FUNCTION_BLOCK MANUAL_PAGE
VAR_INPUT
	STRING_PG1 : STRING;
	STRING_PG2 : STRING;
	STRING_PG3 : STRING;
	STRING_PG4 : STRING;
	STRING_PG5 : STRING;
	STRING_PG6 : STRING;
	STRING_PG7 : STRING;
	STRING_PG8 : STRING;
	STRING_PG9 : STRING;
	STRING_PG10 : STRING;
	STRING_PG11 : STRING;
	STRING_PG12 : STRING;
	STRING_PG13 : STRING;
	STRING_PG14 : STRING;
	STRING_PG15 : STRING;
	STRING_PG16 : STRING;
	STRING_PG17 : STRING;
	STRING_PG18 : STRING;
	STRING_PG19 : STRING;
	STRING_PG20 : STRING;
	STRING_CVISU : STRING;


END_VAR
VAR_OUTPUT
	PG_CONFIRMED_BOOL : BOOL;

END_VAR
VAR
END_VAR

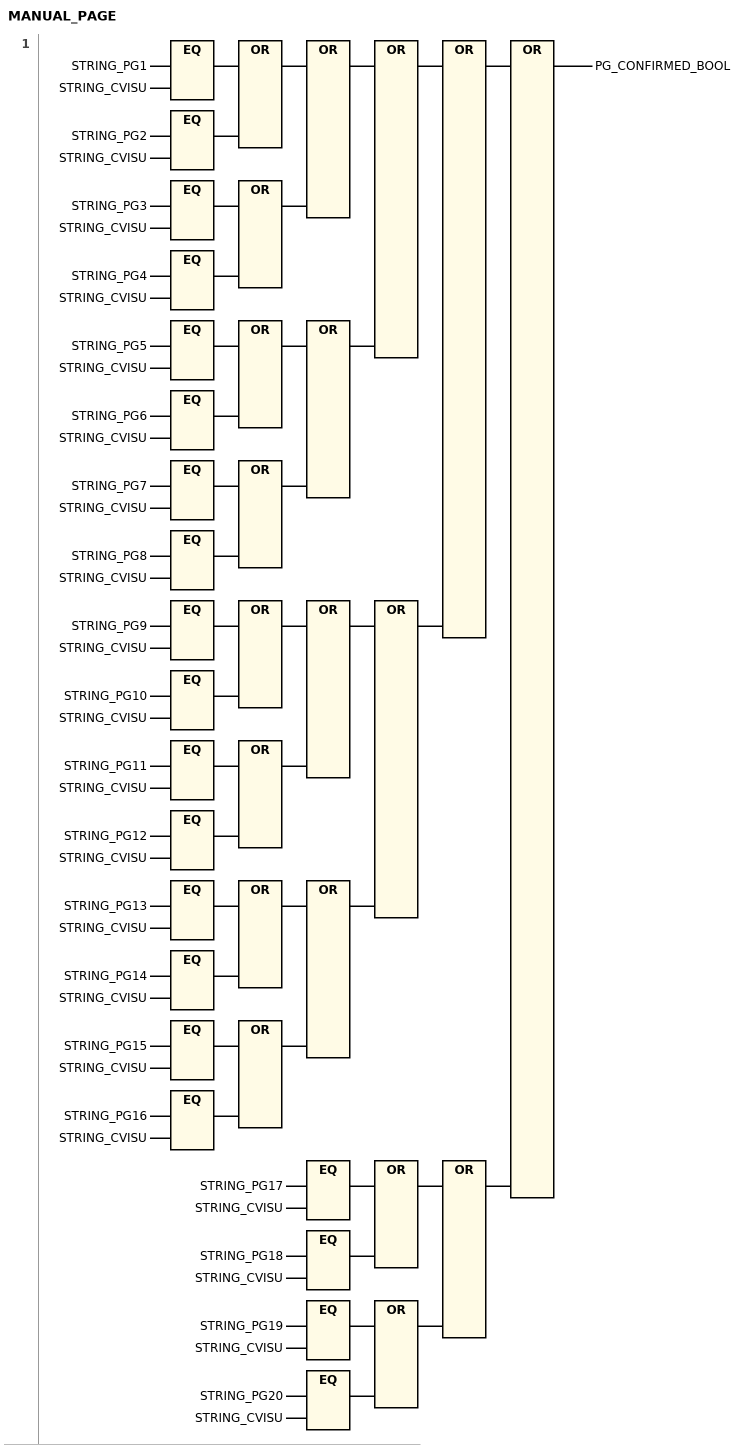
// NETWORK 1
PG_CONFIRMED_BOOL := ((((STRING_PG1 = STRING_CVISU OR STRING_PG2 = STRING_CVISU) OR (STRING_PG3 = STRING_CVISU OR STRING_PG4 = STRING_CVISU)) OR ((STRING_PG5 = STRING_CVISU OR STRING_PG6 = STRING_CVISU) OR (STRING_PG7 = STRING_CVISU OR STRING_PG8 = STRING_CVISU))) OR (((STRING_PG9 = STRING_CVISU OR STRING_PG10 = STRING_CVISU) OR (STRING_PG11 = STRING_CVISU OR STRING_PG12 = STRING_CVISU)) OR ((STRING_PG13 = STRING_CVISU OR STRING_PG14 = STRING_CVISU) OR (STRING_PG15 = STRING_CVISU OR STRING_PG16 = STRING_CVISU)))) OR ((STRING_PG17 = STRING_CVISU OR STRING_PG18 = STRING_CVISU) OR (STRING_PG19 = STRING_CVISU OR STRING_PG20 = STRING_CVISU));

END_FUNCTION_BLOCK

(* stored: Version 1.1.0.1, ProductVersion 3.1.4024.12
   POU MANUAL_PAGE: Id {d8dec126-5e01-4cf6-a0fe-0bff10b5bf3e}, SpecialFunc None *)
